TYPE Roller :
STRUCT
	Power  			: BOOL;
	forward  		: BOOL; 
	backward		: BOOL;
	//run             :BOOL;  //2024.05.26 new added by martin
	//direction       :BOOL;  //2024.05.26 new added by martin
	err 			: FB_DigitalInput;
	sensor 			: FB_DigitalInput;
END_STRUCT
END_TYPE

(* stored: Version 1.1.0.1, ProductVersion 3.1.4024.12
   DUT Roller: Id {2dbdf7ad-cdf6-46d1-abd3-013eeb4d7cf7} *)
